// TIA Portal project "Crossing_FactoryIO" (V14)
// Vorlageprojekt für das Buch mit Zielsystem S7-1200

(* hardware
DEVICE "S7-1200-Station_1"  S7-1200 Station
   slot 0: "Baugruppenträger_0"  Rack  V1.0
   slot 1: "PLC_1"  CPU 1211C DC/DC/DC  6ES7 211-1AE40-0XB0  V4.1
*)

// ===== PLC "PLC_1"  CPU 1211C DC/DC/DC =====

VAR_GLOBAL   // PLC tag table "Standard-Variablentabelle"
   "System_Byte" AT %MB1 : Byte;
   "FirstScan" AT %M1.0 : Bool;
   "DiagStatusUpdate" AT %M1.1 : Bool;
   "AlwaysTRUE" AT %M1.2 : Bool;
   "AlwaysFALSE" AT %M1.3 : Bool;
   "Clock_Byte" AT %MB0 : Byte;
   "Clock_10Hz" AT %M0.0 : Bool;
   "Clock_5Hz" AT %M0.1 : Bool;
   "Clock_2.5Hz" AT %M0.2 : Bool;
   "Clock_2Hz" AT %M0.3 : Bool;
   "Clock_1.25Hz" AT %M0.4 : Bool;
   "Clock_1Hz" AT %M0.5 : Bool;
   "Clock_0.625Hz" AT %M0.6 : Bool;
   "Clock_0.5Hz" AT %M0.7 : Bool;
END_VAR

VAR_GLOBAL   // PLC tag table "Tag_table_crossing"
   "P1" AT %M10.0 : Bool;
   "P2" AT %M10.1 : Bool;
   "PP" AT %MB16 : USInt;
   "TimetoCG" AT %QD30 : DInt;
   "CarTooFast1" AT %M10.4 : Bool;
   "CarTooFast2" AT %M10.5 : Bool;
   "PedestrianButton1" AT %I0.0 : Bool;
   "CarGreen1" AT %Q0.0 : Bool;
   "CarGreen2" AT %Q0.1 : Bool;
   "CarRed1" AT %Q0.2 : Bool;
   "CarRed2" AT %Q0.3 : Bool;
   "CarYellow1" AT %Q0.4 : Bool;
   "CarYellow2" AT %Q0.5 : Bool;
   "PedestrianGreen1" AT %Q0.6 : Bool;
   "PedestrianRed1" AT %Q0.7 : Bool;
   "PedestrianGreen2" AT %Q1.0 : Bool;
   "PedestrianRed2" AT %Q1.1 : Bool;
   "PedestrianButtonPressed" AT %Q1.2 : Bool;
   "PedestrianButton2" AT %I0.1 : Bool;
   "Mode" AT %I0.2 : Bool;
   "ButtonFlt1" AT %I0.3 : Bool;
   "ButtonFlt2" AT %I0.4 : Bool;
   "ResetSystem" AT %I0.5 : Bool;
   "PedestrianButtonPressed2" AT %Q1.3 : Bool;
   "TimetoCG2" AT %QD34 : DInt;
   "ButtonFaultLight" AT %Q1.4 : Bool;
   "ButtonFaultLight 2" AT %Q1.5 : Bool;
   "ModeLight" AT %Q1.6 : Bool;
END_VAR

DATA_BLOCK "FB_Crossing_DB"   // DB1
{ S7_Optimized_Access := 'TRUE' }
VERSION : 0.1
// stored: InstanceOfName FB_Crossing
"FB_Crossing"
BEGIN
END_DATA_BLOCK

FUNCTION_BLOCK "FB_Crossing"   // FB1, LAD
{ S7_Optimized_Access := 'TRUE' }
VERSION : 0.1
   VAR_INPUT
      Pedestrian_1 : Bool;   // signal for a button activated by the first pedestrian.
      Pedestrian_2 : Bool;   // signal for a button activated by the second pedestrian
      SystemStopWhenBroken : Bool;   // 1=YellowBlinking, 0=AutosequenceNtOk
      ResetSystem : Bool;   // signal for resetting the system to its initial state
   END_VAR
   VAR_OUTPUT
      CR : Bool;   // red light for cars
      CY : Bool;   // yellow light for cars
      CG : Bool;   // green light for car
      PG : Bool;   // green light for pedestrians
      PR : Bool;   // red light for pedestrians
      WAIT : USInt;   // Output that could indicate waiting time or waiting status
      TimeForCarGreen : USInt;   // A variable representing the duration for which the green light for cars should stay on
      PedestrianButtonPressed : Bool;   // represent status od sequence pedestrian to green
   END_VAR
   VAR
      "array" : Array[0..10] of Bool;
      Car : Struct
         Red : Bool;
         Yellow : Bool;
         Green : Bool;
      END_STRUCT;
      Pedestrian : Struct
         Red : Bool;
         Green : Bool;
      END_STRUCT;
      Sequence : Struct
         PushButtonPressed : Bool;
         CarRed : Bool;
         PedestrianGreen : Bool;
         PedestrianToBlinking : Bool;
         PedestrianBlinking : Bool;
         CarYellowRed : Bool;
         CarGreen : Bool;
         Blocade : Bool;
      END_STRUCT;
      Timer_CarToYellow : TON_TIME;
      Timer_CarToRed : TON_TIME;
      Timer_PedestrianToGreen : TON_TIME;
      Timer_PedestrianToBlinking : TON_TIME;
      Timer_PedestrianToRed : TON_TIME;
      Timer_CarToYellowRed : TON_TIME;
      Timer_CarToGreen : TON_TIME;
      Timer_blocade : TON_TIME;
      Timer_breakdown : TON_TIME;
      timer_Autoseq_NOT_OK : TON_TIME;
      Timer_Autoseq_OK : TON_TIME;
      Timer_DisplayTimeToCarGreen : TON_TIME;
      SystemStopBroken : Bool;
   END_VAR
   VAR_TEMP
      tmp : Bool;
      TimeToGreen : Time;
      TimeToGreenUDint : DInt;
   END_VAR
   VAR_TEMP   // added for the SCL form of the ladder/FBD networks
      _w1 : Bool;
      _w2 : Bool;
      _w3 : Bool;
   END_VAR
BEGIN

REGION Network 1: init
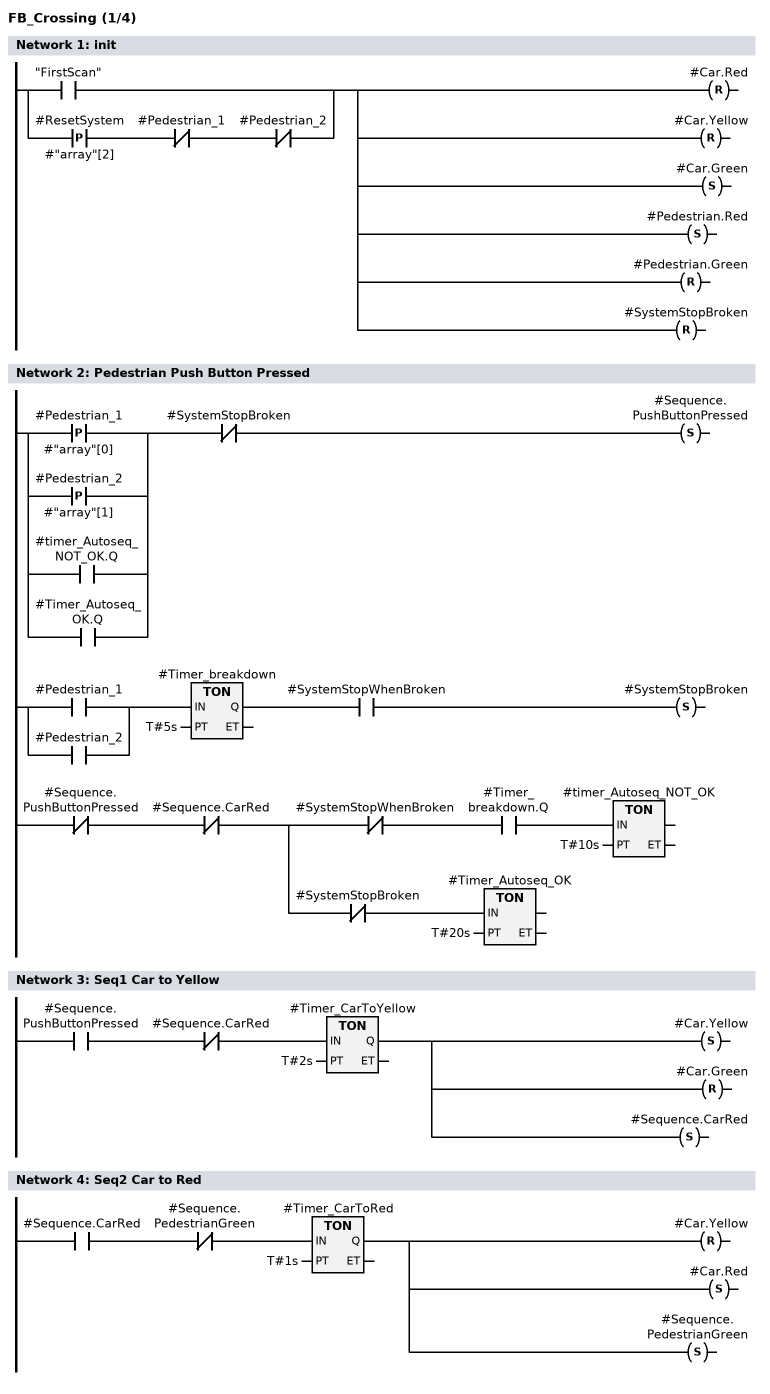
   RUNG wire#powerrail
      Contact( "FirstScan" )
      wire#w1
      R_Coil( #Car.Red )
   END_RUNG
   RUNG wire#powerrail
      P_Contact(operand := #ResetSystem, bit := #"array"[2])
      I_Contact( #Pedestrian_1 )
      I_Contact( #Pedestrian_2 )
   END_RUNG wire#w1
   RUNG wire#w1
      R_Coil( #Car.Yellow )
   END_RUNG
   RUNG wire#w1
      S_Coil( #Car.Green )
   END_RUNG
   RUNG wire#w1
      S_Coil( #Pedestrian.Red )
   END_RUNG
   RUNG wire#w1
      R_Coil( #Pedestrian.Green )
   END_RUNG
   RUNG wire#w1
      R_Coil( #SystemStopBroken )
   END_RUNG
   // the same network as SCL:
   #_w1 := #ResetSystem AND NOT #"array"[2];   // rising edge of #ResetSystem
   #"array"[2] := #ResetSystem;
   IF "FirstScan" OR (#_w1 AND NOT #Pedestrian_1 AND NOT #Pedestrian_2) THEN
       #Car.Red := FALSE;
       #Car.Yellow := FALSE;
       #Car.Green := TRUE;
       #Pedestrian.Red := TRUE;
       #Pedestrian.Green := FALSE;
       #SystemStopBroken := FALSE;
   END_IF;
END_REGION

REGION Network 2: Pedestrian Push Button Pressed
   #_w1 := #Pedestrian_1 AND NOT #"array"[0];   // rising edge of #Pedestrian_1
   #"array"[0] := #Pedestrian_1;
   #_w2 := #Pedestrian_2 AND NOT #"array"[1];   // rising edge of #Pedestrian_2
   #"array"[1] := #Pedestrian_2;
   IF (#_w1 OR #_w2 OR #timer_Autoseq_NOT_OK.Q OR #Timer_Autoseq_OK.Q) AND NOT #SystemStopBroken THEN
       #Sequence.PushButtonPressed := TRUE;
   END_IF;
   #Timer_breakdown(IN := #Pedestrian_1 OR #Pedestrian_2, PT := T#5s);   // TON
   IF #Timer_breakdown.Q AND #SystemStopWhenBroken THEN #SystemStopBroken := TRUE; END_IF;
   #_w3 := NOT #Sequence.PushButtonPressed AND NOT #Sequence.CarRed;
   #timer_Autoseq_NOT_OK(IN := #_w3 AND NOT #SystemStopWhenBroken AND #Timer_breakdown.Q, PT := T#10s);   // TON
   #Timer_Autoseq_OK(IN := #_w3 AND NOT #SystemStopBroken, PT := T#20s);   // TON
END_REGION

REGION Network 3: Seq1 Car to Yellow
   #Timer_CarToYellow(IN := #Sequence.PushButtonPressed AND NOT #Sequence.CarRed, PT := T#2s);   // TON
   IF #Timer_CarToYellow.Q THEN
       #Car.Yellow := TRUE;
       #Car.Green := FALSE;
       #Sequence.CarRed := TRUE;
   END_IF;
END_REGION

REGION Network 4: Seq2 Car to Red
   #Timer_CarToRed(IN := #Sequence.CarRed AND NOT #Sequence.PedestrianGreen, PT := T#1s);   // TON
   IF #Timer_CarToRed.Q THEN
       #Car.Yellow := FALSE;
       #Car.Red := TRUE;
       #Sequence.PedestrianGreen := TRUE;
   END_IF;
END_REGION

REGION Network 5: Seq3 Pedestrian to Green
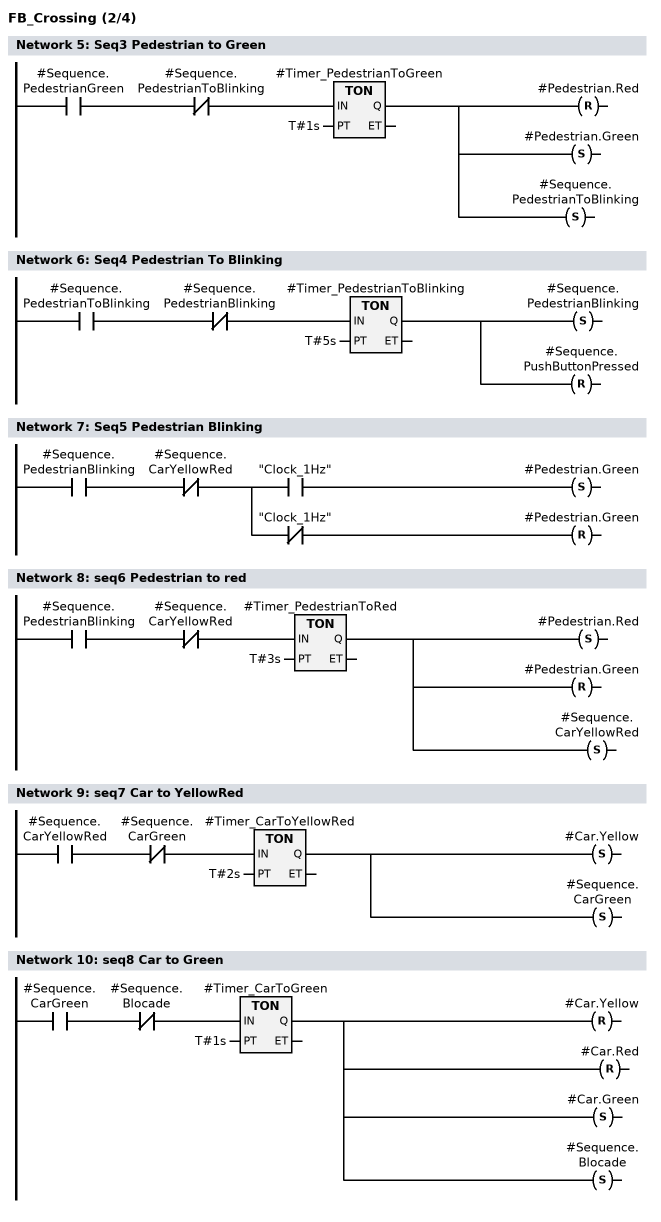
   #Timer_PedestrianToGreen(IN := #Sequence.PedestrianGreen AND NOT #Sequence.PedestrianToBlinking, PT := T#1s);   // TON
   IF #Timer_PedestrianToGreen.Q THEN
       #Pedestrian.Red := FALSE;
       #Pedestrian.Green := TRUE;
       #Sequence.PedestrianToBlinking := TRUE;
   END_IF;
END_REGION

REGION Network 6: Seq4 Pedestrian To Blinking
   #Timer_PedestrianToBlinking(IN := #Sequence.PedestrianToBlinking AND NOT #Sequence.PedestrianBlinking,   // TON
                           PT := T#5s);
   IF #Timer_PedestrianToBlinking.Q THEN
       #Sequence.PedestrianBlinking := TRUE;
       #Sequence.PushButtonPressed := FALSE;
   END_IF;
END_REGION

REGION Network 7: Seq5 Pedestrian Blinking
   RUNG wire#powerrail
      Contact( #Sequence.PedestrianBlinking )
      I_Contact( #Sequence.CarYellowRed )
      wire#w1
      Contact( "Clock_1Hz" )
      S_Coil( #Pedestrian.Green )
   END_RUNG
   RUNG wire#w1
      I_Contact( "Clock_1Hz" )
      R_Coil( #Pedestrian.Green )
   END_RUNG
   // the same network as SCL:
   #_w1 := #Sequence.PedestrianBlinking AND NOT #Sequence.CarYellowRed;
   IF #_w1 AND "Clock_1Hz" THEN #Pedestrian.Green := TRUE; END_IF;
   IF #_w1 AND NOT "Clock_1Hz" THEN #Pedestrian.Green := FALSE; END_IF;
END_REGION

REGION Network 8: seq6 Pedestrian to red
   #Timer_PedestrianToRed(IN := #Sequence.PedestrianBlinking AND NOT #Sequence.CarYellowRed, PT := T#3s);   // TON
   IF #Timer_PedestrianToRed.Q THEN
       #Pedestrian.Red := TRUE;
       #Pedestrian.Green := FALSE;
       #Sequence.CarYellowRed := TRUE;
   END_IF;
END_REGION

REGION Network 9: seq7 Car to YellowRed
   #Timer_CarToYellowRed(IN := #Sequence.CarYellowRed AND NOT #Sequence.CarGreen, PT := T#2s);   // TON
   IF #Timer_CarToYellowRed.Q THEN
       #Car.Yellow := TRUE;
       #Sequence.CarGreen := TRUE;
   END_IF;
END_REGION

REGION Network 10: seq8 Car to Green
   #Timer_CarToGreen(IN := #Sequence.CarGreen AND NOT #Sequence.Blocade, PT := T#1s);   // TON
   IF #Timer_CarToGreen.Q THEN
       #Car.Yellow := FALSE;
       #Car.Red := FALSE;
       #Car.Green := TRUE;
       #Sequence.Blocade := TRUE;
   END_IF;
END_REGION

REGION Network 11: seq9 Blocade
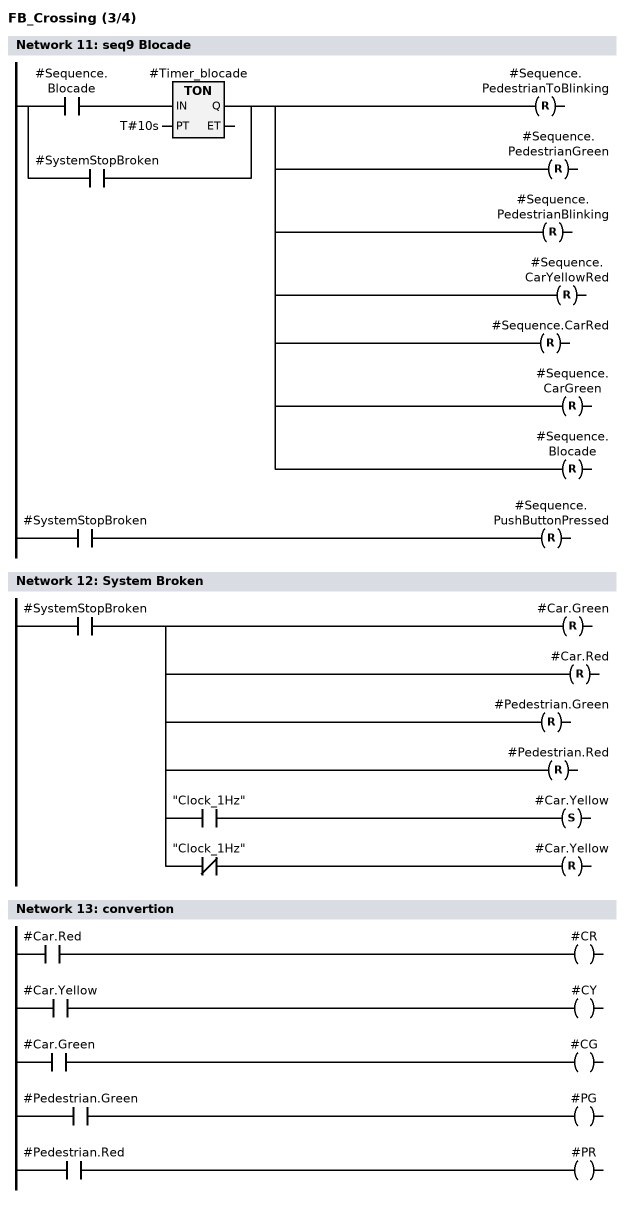
   #Timer_blocade(IN := #Sequence.Blocade, PT := T#10s);   // TON
   IF #Timer_blocade.Q OR #SystemStopBroken THEN
       #Sequence.PedestrianToBlinking := FALSE;
       #Sequence.PedestrianGreen := FALSE;
       #Sequence.PedestrianBlinking := FALSE;
       #Sequence.CarYellowRed := FALSE;
       #Sequence.CarRed := FALSE;
       #Sequence.CarGreen := FALSE;
       #Sequence.Blocade := FALSE;
   END_IF;
   IF #SystemStopBroken THEN #Sequence.PushButtonPressed := FALSE; END_IF;
END_REGION

REGION Network 12: System Broken
   RUNG wire#powerrail
      Contact( #SystemStopBroken )
      wire#w1
      R_Coil( #Car.Green )
   END_RUNG
   RUNG wire#w1
      R_Coil( #Car.Red )
   END_RUNG
   RUNG wire#w1
      R_Coil( #Pedestrian.Green )
   END_RUNG
   RUNG wire#w1
      R_Coil( #Pedestrian.Red )
   END_RUNG
   RUNG wire#w1
      Contact( "Clock_1Hz" )
      S_Coil( #Car.Yellow )
   END_RUNG
   RUNG wire#w1
      I_Contact( "Clock_1Hz" )
      R_Coil( #Car.Yellow )
   END_RUNG
   // the same network as SCL:
   IF #SystemStopBroken THEN
       #Car.Green := FALSE;
       #Car.Red := FALSE;
       #Pedestrian.Green := FALSE;
       #Pedestrian.Red := FALSE;
   END_IF;
   IF #SystemStopBroken AND "Clock_1Hz" THEN #Car.Yellow := TRUE; END_IF;
   IF #SystemStopBroken AND NOT "Clock_1Hz" THEN #Car.Yellow := FALSE; END_IF;
END_REGION

REGION Network 13: convertion
   RUNG wire#powerrail
      Contact( #Car.Red )
      Coil( #CR )
   END_RUNG
   RUNG wire#powerrail
      Contact( #Car.Yellow )
      Coil( #CY )
   END_RUNG
   RUNG wire#powerrail
      Contact( #Car.Green )
      Coil( #CG )
   END_RUNG
   RUNG wire#powerrail
      Contact( #Pedestrian.Green )
      Coil( #PG )
   END_RUNG
   RUNG wire#powerrail
      Contact( #Pedestrian.Red )
      Coil( #PR )
   END_RUNG
   // the same network as SCL:
   #CR := #Car.Red;
   #CY := #Car.Yellow;
   #CG := #Car.Green;
   #PG := #Pedestrian.Green;
   #PR := #Pedestrian.Red;
END_REGION

REGION Network 14: time for car green
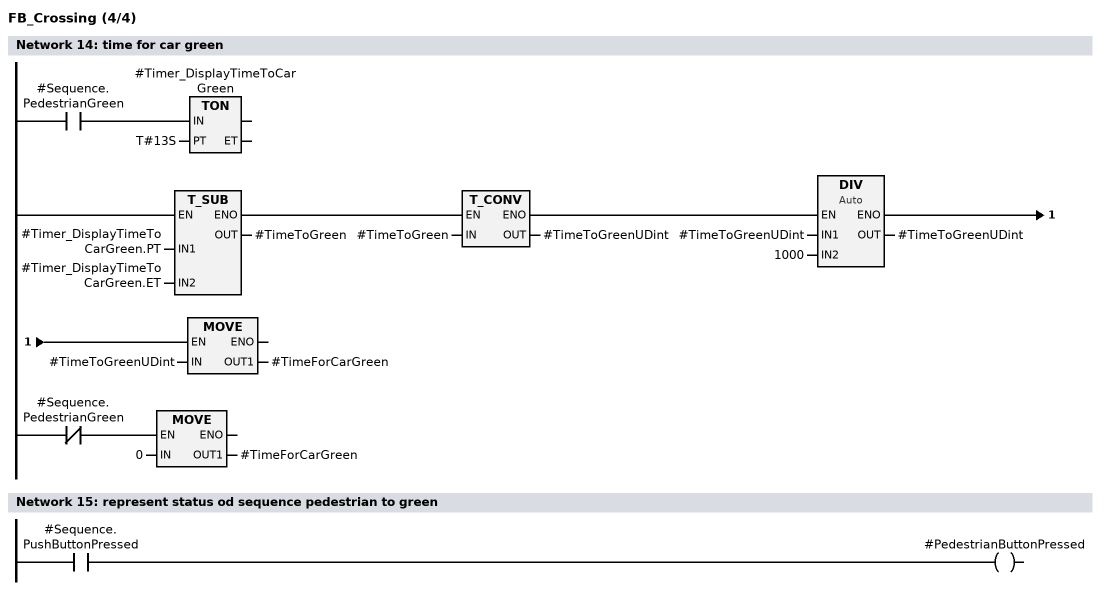
   // ENO of a box is taken as its EN; it also drops when the box reports an error
   #Timer_DisplayTimeToCarGreen(IN := #Sequence.PedestrianGreen, PT := T#13S);   // TON
   #TimeToGreen := T_SUB(IN1 := #Timer_DisplayTimeToCarGreen.PT, IN2 := #Timer_DisplayTimeToCarGreen.ET);
   #TimeToGreenUDint := T_CONV(IN := #TimeToGreen);
   #TimeToGreenUDint := #TimeToGreenUDint / 1000;
   #TimeForCarGreen := #TimeToGreenUDint;
   IF NOT #Sequence.PedestrianGreen THEN #TimeForCarGreen := 0; END_IF;
END_REGION

REGION Network 15: represent status od sequence pedestrian to green
   RUNG wire#powerrail
      Contact( #Sequence.PushButtonPressed )
      Coil( #PedestrianButtonPressed )
   END_RUNG
   // the same network as SCL:
   #PedestrianButtonPressed := #Sequence.PushButtonPressed;
END_REGION
END_FUNCTION_BLOCK

FUNCTION "MHJ-PLC-Lab-Function-S71200" : Void   // FC9000, SCL
{ S7_Optimized_Access := 'TRUE' }
VERSION : 0.1
   VAR_TEMP
      rdTimeReturn : Int;
      outputTime : DTL;
      SyncVal : Byte;
      forVal : Int;
      forVal_2 : Int;
      Value : Byte;
   END_VAR
   VAR CONSTANT
      CompVal : Byte := 16#34;
      Value_01 : Byte := 16#11;
      Value_01_DW : DWord := 16#A165_D992;
      Value_02_DW : DWord := 16#58BE_4401;
   END_VAR
BEGIN

   #Value:=PEEK(area := 16#82,
        dbNumber := 0,
        byteOffset := 511);
   #Value := #Value + 1;

   POKE(area := 16#82,
        dbNumber := 0,
        byteOffset := 511,
        value := #Value);

   POKE(area:=16#81,
        dbNumber:=0,
        byteOffset:=1016,
        value:=#Value_01_DW);
   POKE(area := 16#81,
        dbNumber := 0,
        byteOffset := 1020,
        value := #Value_02_DW);

   POKE(area := 16#81,
        dbNumber := 0,
        byteOffset := 511,
        value := B#16#00);

   FOR #forVal := 0 TO 120 DO
       FOR #forVal_2:=0 TO 10 DO
           #rdTimeReturn:=RD_SYS_T(#outputTime);
           #rdTimeReturn := WR_SYS_T(#outputTime);
           #rdTimeReturn := RD_SYS_T(#outputTime);
           #rdTimeReturn := WR_SYS_T(#outputTime);
       END_FOR;
       #SyncVal:= PEEK(area := 16#81,
                      dbNumber := 0,
                      byteOffset := 511);
       IF #SyncVal = #CompVal THEN
          GOTO M_1;
       END_IF;
   END_FOR;
   RETURN;

   M_1:
   POKE(area := 16#81,
        dbNumber := 0,
        byteOffset := 511,
        value := B#16#0);
END_FUNCTION

ORGANIZATION_BLOCK "Main"   // OB1, LAD, ProgramCycle
TITLE = "Main Program Sweep (Cycle)"
{ S7_Optimized_Access := 'TRUE' }
VERSION : 0.1
   VAR_INPUT
      Initial_Call : Bool;   // Initial call of this OB
      Remanence : Bool;   // =True, if remanent data are available
   END_VAR
   VAR_TEMP
      "WWW_RET_VAL Int" : Bool;
   END_VAR
BEGIN

REGION Network 1: Konnektierungsbaustein für PLC-Lab / FactoryIO communication
   // Im Netzwerk 1 wird der Konnektierungsbaustein für PLC-Lab aufgerufen.
   // Dieser Aufruf darf nicht entfernt werden!
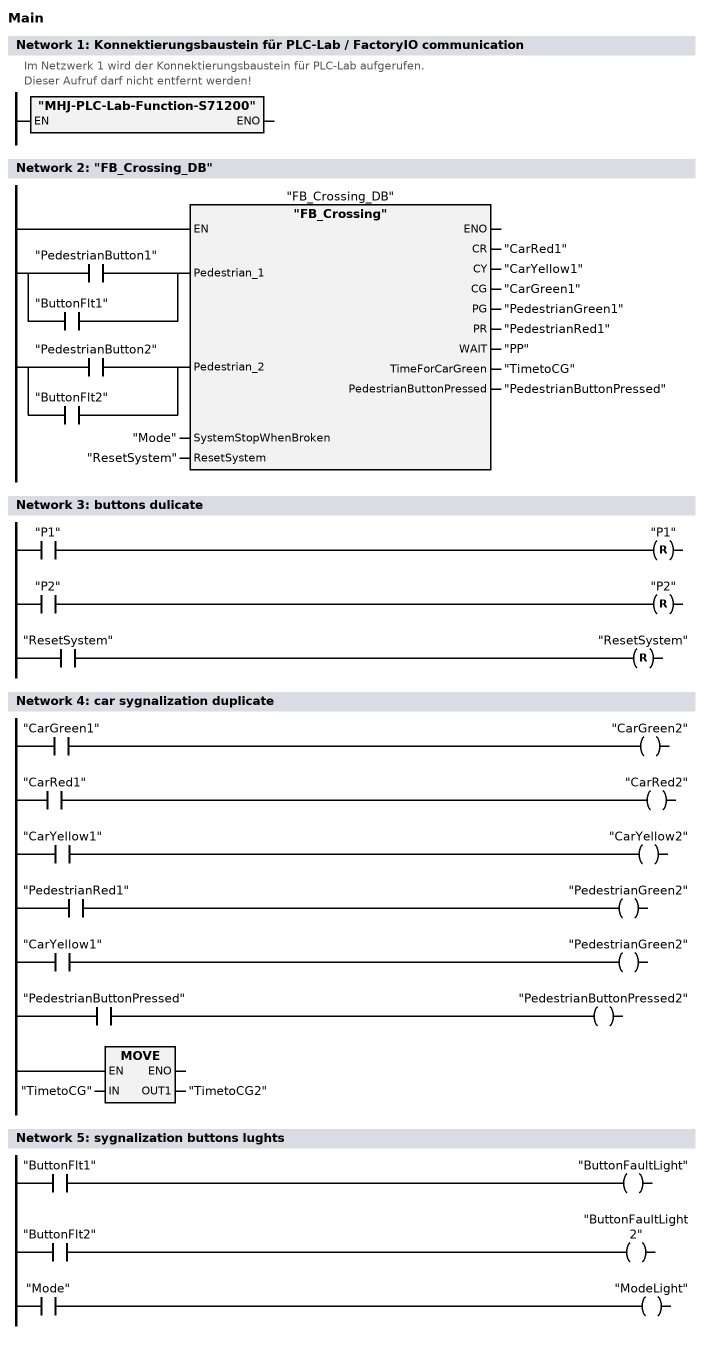
   RUNG wire#powerrail
      "MHJ-PLC-Lab-Function-S71200"()
   END_RUNG
   // the same network as SCL:
   "MHJ-PLC-Lab-Function-S71200"();
END_REGION

REGION Network 2: "FB_Crossing_DB"
   RUNG wire#powerrail
      "FB_Crossing_DB"(Pedestrian_1 := wire#w1, Pedestrian_2 := wire#w2, SystemStopWhenBroken := "Mode", ResetSystem := "ResetSystem", CR => "CarRed1", CY => "CarYellow1", CG => "CarGreen1", PG => "PedestrianGreen1", PR => "PedestrianRed1", WAIT => "PP", TimeForCarGreen => "TimetoCG", PedestrianButtonPressed => "PedestrianButtonPressed")
   END_RUNG
   RUNG wire#powerrail
      Contact( "PedestrianButton1" )
   END_RUNG wire#w1
   RUNG wire#powerrail
      Contact( "ButtonFlt1" )
   END_RUNG wire#w1
   RUNG wire#powerrail
      Contact( "PedestrianButton2" )
   END_RUNG wire#w2
   RUNG wire#powerrail
      Contact( "ButtonFlt2" )
   END_RUNG wire#w2
   // the same network as SCL:
   "FB_Crossing_DB"(Pedestrian_1 := "PedestrianButton1" OR "ButtonFlt1",   // "FB_Crossing"
                    Pedestrian_2 := "PedestrianButton2" OR "ButtonFlt2",
                    SystemStopWhenBroken := "Mode",
                    ResetSystem := "ResetSystem",
                    CR => "CarRed1",
                    CY => "CarYellow1",
                    CG => "CarGreen1",
                    PG => "PedestrianGreen1",
                    PR => "PedestrianRed1",
                    WAIT => "PP",
                    TimeForCarGreen => "TimetoCG",
                    PedestrianButtonPressed => "PedestrianButtonPressed");
END_REGION

REGION Network 3: buttons dulicate
   RUNG wire#powerrail
      Contact( "P1" )
      R_Coil( "P1" )
   END_RUNG
   RUNG wire#powerrail
      Contact( "P2" )
      R_Coil( "P2" )
   END_RUNG
   RUNG wire#powerrail
      Contact( "ResetSystem" )
      R_Coil( "ResetSystem" )
   END_RUNG
   // the same network as SCL:
   IF "P1" THEN "P1" := FALSE; END_IF;
   IF "P2" THEN "P2" := FALSE; END_IF;
   IF "ResetSystem" THEN "ResetSystem" := FALSE; END_IF;
END_REGION

REGION Network 4: car sygnalization duplicate
   RUNG wire#powerrail
      Contact( "CarGreen1" )
      Coil( "CarGreen2" )
   END_RUNG
   RUNG wire#powerrail
      Contact( "CarRed1" )
      Coil( "CarRed2" )
   END_RUNG
   RUNG wire#powerrail
      Contact( "CarYellow1" )
      Coil( "CarYellow2" )
   END_RUNG
   RUNG wire#powerrail
      Contact( "PedestrianRed1" )
      Coil( "PedestrianGreen2" )
   END_RUNG
   RUNG wire#powerrail
      Contact( "CarYellow1" )
      Coil( "PedestrianGreen2" )
   END_RUNG
   RUNG wire#powerrail
      Contact( "PedestrianButtonPressed" )
      Coil( "PedestrianButtonPressed2" )
   END_RUNG
   RUNG wire#powerrail
      Move(in := "TimetoCG", out1 => "TimetoCG2")
   END_RUNG
   // the same network as SCL:
   "CarGreen2" := "CarGreen1";
   "CarRed2" := "CarRed1";
   "CarYellow2" := "CarYellow1";
   "PedestrianGreen2" := "PedestrianRed1";
   "PedestrianGreen2" := "CarYellow1";
   "PedestrianButtonPressed2" := "PedestrianButtonPressed";
   "TimetoCG2" := "TimetoCG";
END_REGION

REGION Network 5: sygnalization buttons lughts
   RUNG wire#powerrail
      Contact( "ButtonFlt1" )
      Coil( "ButtonFaultLight" )
   END_RUNG
   RUNG wire#powerrail
      Contact( "ButtonFlt2" )
      Coil( "ButtonFaultLight 2" )
   END_RUNG
   RUNG wire#powerrail
      Contact( "Mode" )
      Coil( "ModeLight" )
   END_RUNG
   // the same network as SCL:
   "ButtonFaultLight" := "ButtonFlt1";
   "ButtonFaultLight 2" := "ButtonFlt2";
   "ModeLight" := "Mode";
END_REGION
END_ORGANIZATION_BLOCK